FUNCTION_BLOCK FB_System_HO_961
VAR_INPUT
	Freigabe_WW_auto			: BOOL;
	Freigabe_HW_auto			: BOOL;
	Betrieb_Anford_WW_auto		: BOOL;
	Betrieb_Anford_HW_auto		: BOOL;
	Freigabe_Deakt_WW_auto		: BOOL;
	Freigabe_Deakt_HW_auto		: BOOL;
END_VAR
VAR_OUTPUT
END_VAR
VAR
	Haerteofen_961						: FB_HO;
	System_Haerteofen_Warmwasser_261	: FB_System_HOWW_261;
	System_Haerteofen_Heisswasser_361	: FB_System_HOHW_361;
END_VAR

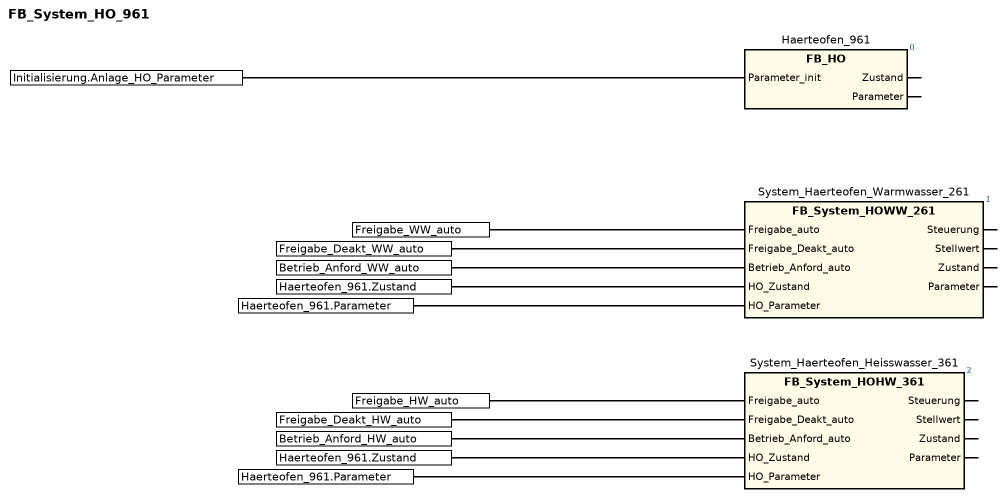
Haerteofen_961(Parameter_init := Initialisierung.Anlage_HO_Parameter); // FB_HO
System_Haerteofen_Warmwasser_261(
    Freigabe_auto := Freigabe_WW_auto,
    Freigabe_Deakt_auto := Freigabe_Deakt_WW_auto,
    Betrieb_Anford_auto := Betrieb_Anford_WW_auto,
    HO_Zustand := Haerteofen_961.Zustand,
    HO_Parameter := Haerteofen_961.Parameter); // FB_System_HOWW_261
System_Haerteofen_Heisswasser_361(
    Freigabe_auto := Freigabe_HW_auto,
    Freigabe_Deakt_auto := Freigabe_Deakt_HW_auto,
    Betrieb_Anford_auto := Betrieb_Anford_HW_auto,
    HO_Zustand := Haerteofen_961.Zustand,
    HO_Parameter := Haerteofen_961.Parameter); // FB_System_HOHW_361

END_FUNCTION_BLOCK

(* stored: Version 1.1.0.1, ProductVersion 3.1.4024.9
   POU FB_System_HO_961: Id {4accc103-5601-42d5-b392-6abd7b19f976}, SpecialFunc None *)
